FUNCTION_BLOCK fbEcCoESdoRead
VAR_INPUT
END_VAR
VAR_OUTPUT
END_VAR
VAR

	FB_EcCoESdoRead: FB_EcCoESdoRead;
END_VAR

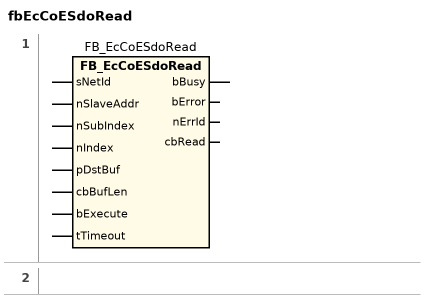
// NETWORK 1
FB_EcCoESdoRead();

// NETWORK 2

END_FUNCTION_BLOCK

(* stored: Version 1.1.0.1, ProductVersion 3.1.4024.12
   POU fbEcCoESdoRead: Id {3b103599-2394-446e-bb14-0f0e22be8be5}, SpecialFunc None *)
